# EPICS substitutions: db/Beckhoff_4XXX/ecmcEL4134.substitutions
file "ecmc_analogOutput-chX.template"
{
  pattern {CH_ID, LINR, ESLO, EOFF, EGU, PREC, LOW, LOLO, HIGH, HIHI, HYST, LLSV, LSV, HSV, HHSV, DRVL, DRVH}
          {01, "SLOPE", "${_ESLO=3.0518509476E-4}", "${_EOFF=0}", "${_EGU=V}", "${_PREC=3}", -10, -10, 10, 10, 0, "MAJOR", "MINOR", "MINOR", "MAJOR", -10, 10}
          {02, "SLOPE", "${_ESLO=3.0518509476E-4}", "${_EOFF=0}", "${_EGU=V}", "${_PREC=3}", -10, -10, 10, 10, 0, "MAJOR", "MINOR", "MINOR", "MAJOR", -10, 10}
          {03, "SLOPE", "${_ESLO=3.0518509476E-4}", "${_EOFF=0}", "${_EGU=V}", "${_PREC=3}", -10, -10, 10, 10, 0, "MAJOR", "MINOR", "MINOR", "MAJOR", -10, 10}
          {04, "SLOPE", "${_ESLO=3.0518509476E-4}", "${_EOFF=0}", "${_EGU=V}", "${_PREC=3}", -10, -10, 10, 10, 0, "MAJOR", "MINOR", "MINOR", "MAJOR", -10, 10}
}
